Universal Robots PolyScope program: b_base0.urp

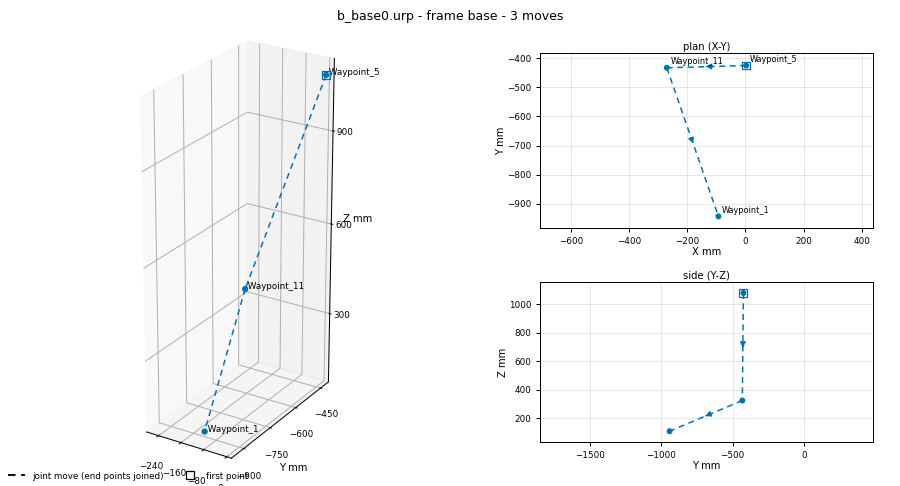
[picture p0: tool path of b_base0.urp in frame base, 3 of 3 moves have a stored position in this frame; points joined in program order, loops and branches not executed]
Program b_base0 (installation=default directory=/programs/Burkat_U_Plant createdIn=5.12.6.1102099 lastSavedIn=5.12.6.1102099 robotSerialNumber=20215500597)
Calibrated DH parameters: a=[0.000193, -0.066673, -0.391568, -0.000012, 0.00005, 0]; d=[0.162643, -472.05677, 465.132521, 7.058239, 0.099746, 0.099582]; alpha=[1.571116, 0.00089, 0.003862, 1.569269, -1.569248, 0]; deltaTheta=[0, -1.413394, 7.628392, 0.068187, 0, -0.000001]
Robot Program (runOnlyOnce=true)
  MoveJ speed 60 deg/s, acceleration 80 deg/s^2 (useActiveTCP=true) feature=Base
    Waypoint Waypoint_5: TCP in base x=2.907 y=-424.808 z=1080.56 mm, rx=-0.0058 ry=2.215 rz=-2.2169 rad; joints [0.172, -90.171, 0.225, -89.838, 0.52, -0.053] deg; TCP offset x=0 y=0 z=191.5 mm, rx=0 ry=0 rz=0 rad
  MoveJ speed 60 deg/s, acceleration 80 deg/s^2 (useActiveTCP=true) feature=Base
    Waypoint Waypoint_11: TCP in base x=-269.994 y=-432.539 z=325.272 mm, rx=1.6722 ry=-0.6368 rz=-0.3794 rad; joints [26.737, -115.333, 124.939, 3.276, 63.256, -0.008] deg
  MoveJ speed 60 deg/s, acceleration 80 deg/s^2 (useActiveTCP=true) feature=Base
    Waypoint Waypoint_1: TCP in base x=-92.58 y=-943.208 z=109.706 mm, rx=1.5938 ry=0.0536 rz=-0.0777 rad; joints [70.625, -40.487, 74.961, -33.19, 71.628, -5.097] deg
  URCap Gripper Activate (Robotiq_Grippers, Robotiq Inc.) dataModel(ResetAndActivateKey=false)
